Staubli VAL3: setOnline.pgx

public program setOnline(num x_nCamID (dimensions=1), bool x_bOnline (dimensions=1), bool& x_bError[] (dimensions=1))
begin
  //-----------------------------------------------------------------------
  //Header begin
  //Description of program
  //  Sets the In-Sight sensor into Online or Offline mode.
  //
  //Input parameters
  //  num x_nCamID :
  //    role :
  //  bool x_bOnline  :
  //    role : if true put camera online otherwise put camera to offline.
  //
  //Output parameters
  //  bool x_bError :
  //    role : returns true if an error occurred and false otherwise
  //
  //Examples
  //  call setOnline(nCamID,"true",l_bError)
  //
  //History
  //  Creation : 19-05-08 - f.Rob
  //Header end
  //-----------------------------------------------------------------------

  nProgram[x_nCamID]=2
  if x_bOnline
    //Sets the In-Sight sensor Online.
    call sendCommand(x_nCamID,"SO1",x_bError)
  else
    //Sets the In-Sight sensor Offline.
    call sendCommand(x_nCamID,"SO0",x_bError)
  endIf
end
